{attribute 'linkalways'}
{attribute 'hide_all_locals'}
FUNCTION_BLOCK ValueReal EXTENDS ValueRealRead IMPLEMENTS Value
VAR
END_VAR

METHOD SetFromType : BOOL
VAR_INPUT
	source : __SYSTEM.AnyType;
END_VAR
SetFromType := ConvertAnyType(source, thisAnyType);
END_METHOD

METHOD SetFromString : BOOL
VAR_INPUT
	value : T_MaxString;
END_VAR
thisValue := STRING_TO_REAL(value);

SetFromString := TRUE;
END_METHOD

METHOD Set : BOOL
VAR_INPUT
	source : ANY;
END_VAR
Set := ConvertAnyType(source, thisAnyType);
END_METHOD

END_FUNCTION_BLOCK

(* stored: Version 1.1.0.1
   POU ValueReal: Id {a30aa23e-9c1c-4dd1-8e9f-3826886ad362}, SpecialFunc None
   Method SetFromType: Id {9de98910-a627-4d7e-a9ab-896dfd7416ae}
   Method SetFromString: Id {90ebc12f-bc26-4f93-bfa6-e3c96ec3cc7a}
   Method Set: Id {a8589a4d-8ee1-4a47-a84e-739238f75d18} *)
